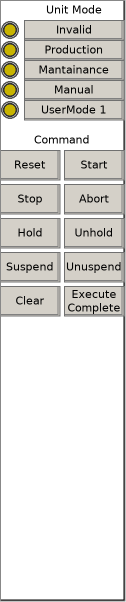
VISUALIZATION VIS_TemplateCommand  // 126x602
VAR_IN_OUT
	eModeCommand	: DINT;
	eStateCommand	: DINT;
	eModeStatus		: DINT;
	eStateStatus	: DINT;
	bModeChangeReq	: BOOL;
END_VAR
    Rectangle (0,0 124x600)
    Lamp1 (0,20 20x20), variable: (eModeStatus = 0), style: Lamp-Lamp1-Yellow
    Button (24,20 100x20), "Invalid", colour toggle: (eModeStatus = 0)
        tap bModeChangeReq
        OnMouseClick: execute { eModeCommand := 0; }
    Lamp1 (0,40 20x20), variable: (eModeStatus = 1), style: Lamp-Lamp1-Yellow
    Button (24,40 100x20), "Production"
        tap bModeChangeReq
        OnMouseClick: execute { eModeCommand := 1; }
    Lamp1 (0,60 20x20), variable: (eModeStatus = 2), style: Lamp-Lamp1-Yellow
    Button (24,60 100x20), "Mantainance"
        tap bModeChangeReq
        OnMouseClick: execute { eModeCommand := 2; }
    Lamp1 (0,80 20x20), variable: (eModeStatus = 3), style: Lamp-Lamp1-Yellow
    Button (24,80 100x20), "Manual"
        tap bModeChangeReq
        OnMouseClick: execute { eModeCommand := 3; }
    Lamp1 (0,100 20x20), variable: (eModeStatus = 4), style: Lamp-Lamp1-Yellow
    Button (24,100 100x20), "UserMode 1"
        tap bModeChangeReq
        OnMouseClick: execute { eModeCommand := 4; }
    Button (0,150 60x30), "Reset"
        OnMouseClick: execute { eStateCommand := 1; }
    Button (64,150 60x30), "Start"
        OnMouseClick: execute { eStateCommand := 2; }
    Button (0,184 60x30), "Stop"
        OnMouseClick: execute { eStateCommand := 3; }
    Button (0,218 60x30), "Hold"
        OnMouseClick: execute { eStateCommand := 4; }
    Button (64,218 60x30), "Unhold"
        OnMouseClick: execute { eStateCommand := 5; }
    Button (0,252 60x30), "Suspend"
        OnMouseClick: execute { eStateCommand := 6; }
    Button (64,252 60x30), "Unuspend"
        OnMouseClick: execute { eStateCommand := 7; }
    Button (0,286 60x30), "Clear"
        OnMouseClick: execute { eStateCommand := 9; }
    Label (0,130 124x20), "Command"
    Button (64,184 60x30), "Abort"
        OnMouseClick: execute { eStateCommand := 8; }
    Button (64,286 60x30), "Execute Complete"
        OnMouseClick: execute { MAIN.bExecuteComplete := TRUE; }
    Label (24,0 100x20), "Unit Mode"
END_VISUALIZATION

(* stored: Version 1.1.0.1
   Visu VIS_TemplateCommand: Id {d7925750-20c5-4482-a15b-9b1c5b9b40e3} *)
